FUNCTION_BLOCK BacnetQD (* Output service interface function block for bacnet double word output data *)
  (* Version 1.0, 2020-01-30, Alexander Tepaev *)
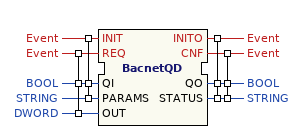
  EVENT_INPUT
    INIT WITH QI, PARAMS; (* Service Initialization *)
    REQ WITH QI, OUT; (* Service Request *)
  END_EVENT
  EVENT_OUTPUT
    INITO WITH QO, STATUS; (* Initialization Confirm *)
    CNF WITH QO, STATUS; (* Confirmation of Requested Service *)
  END_EVENT
  VAR_INPUT
    QI : BOOL; (* Event Input Qualifier *)
    PARAMS : STRING; (* Service Parameters *)
    OUT : DWORD; (* Output data to resource *)
  END_VAR
  VAR_OUTPUT
    QO : BOOL; (* Event Output Qualifier *)
    STATUS : STRING; (* Service Status *)
  END_VAR
END_FUNCTION_BLOCK
